// TIA Portal project "SistemaDePortaDeGaragem" (V16)

(* hardware
DEVICE "S7-1200 station_1"  S7-1200 Station
   slot 0: "Rack_0"  S7-1200 Rack  Rack  V1.0
   slot 1: "PLC_1"  CPU 1214C DC/DC/DC  6ES7 214-1AG40-0XB0  V4.4
DEVICE "HMI_1"  KTP1000 Basic color PN
   slot 0: "HMI_1"  KTP1000 Basic color PN  6AV6 647-0AF11-3AX0  12.0.0.0
   slot 1: "HMI_RT_1"  KTP1000 Basic color PN  6AV6 647-0AF11-3AX0  12.0.0.0
   slot 5: "HMI_1.IE_CP_1"  PROFINET Interface  12.0.0.0
      slot 1: "PROFINET Interface_1"  PROFINET Interface
         slot 1: "Port_1"  Port
*)

// ===== PLC "PLC_1"  CPU 1214C DC/DC/DC =====

VAR_GLOBAL   // PLC tag table "Default tag table"
   "System_Byte" AT %MB1 : Byte;
   "FirstScan" AT %M1.0 : Bool;
   "DiagStatusUpdate" AT %M1.1 : Bool;
   "AlwaysTRUE" AT %M1.2 : Bool;
   "AlwaysFALSE" AT %M1.3 : Bool;
   "Clock_Byte" AT %MB0 : Byte;
   "Clock_10Hz" AT %M0.0 : Bool;
   "Clock_5Hz" AT %M0.1 : Bool;
   "Clock_2.5Hz" AT %M0.2 : Bool;
   "Clock_2Hz" AT %M0.3 : Bool;
   "Clock_1.25Hz" AT %M0.4 : Bool;
   "Clock_1Hz" AT %M0.5 : Bool;
   "Clock_0.625Hz" AT %M0.6 : Bool;
   "Clock_0.5Hz" AT %M0.7 : Bool;
   "BotaoAbrir" AT %I0.1 : Bool;
   "BotaoFechar" AT %I0.2 : Bool;
   "SensorPortaAberta" AT %I0.3 : Bool;
   "SensorPortaFechada" AT %I0.4 : Bool;
   "SensorInfravermelho" AT %I0.5 : Bool;
   "MotorAbrirPortao" AT %Q0.1 : Bool;
   "MotorFecharPortao" AT %Q0.2 : Bool;
END_VAR

FUNCTION "ControlaPortao" : Void   // FC1, LAD
{ S7_Optimized_Access := 'TRUE' }
VERSION : 0.1
BEGIN

REGION Network 1
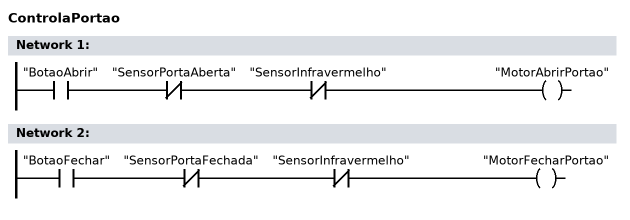
   RUNG wire#powerrail
      Contact( "BotaoAbrir" )
      I_Contact( "SensorPortaAberta" )
      I_Contact( "SensorInfravermelho" )
      Coil( "MotorAbrirPortao" )
   END_RUNG
   // the same network as SCL:
   "MotorAbrirPortao" := "BotaoAbrir" AND NOT "SensorPortaAberta" AND NOT "SensorInfravermelho";
END_REGION

REGION Network 2
   RUNG wire#powerrail
      Contact( "BotaoFechar" )
      I_Contact( "SensorPortaFechada" )
      I_Contact( "SensorInfravermelho" )
      Coil( "MotorFecharPortao" )
   END_RUNG
   // the same network as SCL:
   "MotorFecharPortao" := "BotaoFechar" AND NOT "SensorPortaFechada" AND NOT "SensorInfravermelho";
END_REGION
END_FUNCTION

ORGANIZATION_BLOCK "Main"   // OB1, LAD, ProgramCycle
TITLE = "Main Program Sweep (Cycle)"
{ S7_Optimized_Access := 'TRUE' }
VERSION : 0.1
   VAR_INPUT
      Initial_Call : Bool;   // Initial call of this OB
      Remanence : Bool;   // =True, if remanent data are available
   END_VAR
BEGIN
END_ORGANIZATION_BLOCK

(* ===== HMI "HMI_RT_1" =====
system functions are stored by id; their names below are inferred from use

HMI tags "Default tag table"
   "Tag_ScreenNumber" : UInt, internal

Template "Template_1" 640x480
   Button "Template_Button" at 560,422 size 79x57; TextOff 'Text'
   Button "Template_Button_1" at 480,422 size 79x57; TextOff 'Text'
   Button "Template_Button_2" at 400,422 size 79x57; TextOff 'Text'
   Button "Template_Button_3" at 320,422 size 79x57; TextOff 'Text'
   Button "Template_Button_4" at 240,422 size 79x57; TextOff 'Text'
   Button "Template_Button_5" at 160,422 size 79x57; TextOff 'Text'
   Button "Alarms" at 80,422 size 79x57; TextOff 'Alarms'; PictureOff "AlarmDisplay_KTP1000_Basic_color_PN"; PictureOn "AlarmDisplay_KTP1000_Basic_color_PN"
      on Release: function_ef3f5d25("Alarm window_Unacknowledged", -1)
   Button "Template_Button_6" at 0,422 size 79x57; TextOff 'Text'
   SymbolicIOField "Symbolic_IO_Field_Screen" at 105,11 size 428x34; TextOff '0'; TextOn '1'; TextList "TextList_ScreenNames"
      ProcessValue <- "Tag_ScreenNumber"
      on Change: ActivateScreenByNumber("Tag_ScreenNumber", 0)
   DateTimeField "HmiScreenItemData" at 535,29 size 105x29
   DateTimeField "HmiScreenItemData_1" at 535,0 size 105x29
   GraphicView "Logo" at 0,0 size 103x58; Picture "Logo of HMI_1"

screen "Root screen" 640x480, template "Template_1"
   on GenerateScreen: SetTag("Tag_ScreenNumber", 1)
   TextField "HmiScreenItemData" at 64,226 size 512x22; Text 'Welcome to HMI_1 (KTP1000 Basic color PN)!'

screen "Screen_1" 640x480
   GraphicView "Graphic view_1" at 302,32 size 309x325; Picture "964743"
   Button "Button_2" at 29,410 size 127x42; TextOff 'Fechar Porta'
   Button "Button_1" at 29,356 size 127x42; TextOff 'Abrir Porta'
   Switch "Switch_1" at 236,100 size 64x32; CaptionText 'Switch'; TextOff 'OFF'; TextOn 'ON'
   TextField "Text field_1" at 166,80 size 137x18; Text 'Sensor Porta Aberta'
   Switch "Switch_2" at 236,308 size 64x32; TextOn 'ON'; CaptionText 'Switch'; TextOff 'OFF'
   TextField "Text field_2" at 159,287 size 144x18; Text 'Sensor Porta Fechada'
   Switch "Switch_3" at 237,200 size 64x32; TextOn 'ON'; CaptionText 'Switch'; TextOff 'OFF'
   TextField "Text field_3" at 161,179 size 140x18; Text 'Sensor de Segurança'
   GraphicView "Graphic view_2" at 301,380 size 186x82; Picture "Graphic_1"
   GraphicView "Graphic view_3" at 512,372 size 96x94; Picture "Eo_circle_green_arrow-up.svg"
   GraphicView "Graphic view_4" at 512,371 size 96x94; Picture "Eo_circle_red_arrow-down.svg"
*)